FUNCTION INTERNAL _FindBestChunk : Results.Result
VAR_INPUT
	nRequesterId		: UDINT;
    nRequestedSize     	: UDINT;
END_VAR
VAR_OUTPUT
    nNewId             	: UDINT;
    nNewSize            : UDINT;
END_VAR
VAR
	i					: UDINT;
	j					: UDINT;
END_VAR

FOR i := 1 TO Param.nChannelSize DO
	IF _Channel.stEntry[i].iSignal <> 0 AND_THEN _Channel.stEntry[i].iSignal.id <> nRequesterId THEN
		i := _Channel.stEntry[i].iSignal.id + _Channel.stEntry[i].iSignal.size - 1;
	ELSE
		FOR j := 0 TO Param.nChannelSize DO
			IF _Channel.stEntry[i + j].iSignal <> 0 AND_THEN _Channel.stEntry[i].iSignal.id <> nRequesterId THEN
				EXIT;
			ELSIF Param.nChannelSize <= i + j THEN
				EXIT;
			END_IF			
		END_FOR
		IF nNewSize = 0 THEN
			nNewId := i;
			nNewSize := j + 1;
		ELSIF  nRequestedSize <= j + 1 AND_THEN nNewSize > j + 1 THEN
			nNewId := i;
			nNewSize := nRequestedSize;
		END_IF
		IF _Channel.stEntry[i + j].iSignal = 0 THEN
			i := i + j;
		ELSE
			i := i + j - 1;
		END_IF
		
	END_IF
END_FOR

IF nNewSize > 0 THEN
	nNewSize := nRequestedSize;
	_FindBestChunk := Results.Ok;
ELSE
	_FindBestChunk := Results.Error;
END_IF

END_FUNCTION

(* stored: Version 1.1.0.1
   POU _FindBestChunk: Id {bf0a026d-cc31-407d-ac75-2d22528103ba}, SpecialFunc None *)
